{attribute addProperty BoxType "EL3356-0030-0025"}
{attribute addProperty Id "ValueAT %I*DINT324"}
{attribute addProperty CRC "525818199"}
{attribute addProperty SizeInBites "32"}
{attribute addProperty SizeInBytes "4"}
TYPE RMB_Value_INT_1F575957 :
STRUCT
	{attribute addProperty Name "Value"}
	Value AT %I* : DINT;
END_STRUCT
END_TYPE

(* stored: Version 1.2.0.0, ProductVersion 3.1.4024.9
   DUT RMB_Value_INT_1F575957: Id {9abf0836-af7c-4247-a97c-1fee8c6968b0} *)
